// TIA Portal V15.1 export
// export: Created 2024-05-17T05:38:21.4668831Z, ExportSetting WithDefaults, DisplayName Totally Integrated Automation Portal, DisplayVersion V15.1 Update 5, DisplayName TIA Portal Openness, DisplayVersion V15.1 Update 5, DisplayName SINAMICS Startdrive Advanced, DisplayVersion V15.1, DisplayName G130, G150, S120, S150, SINAMICS MV, S210, DisplayVersion V15.1, DisplayName G110M, G120, G120C, G120D, G120P, DisplayVersion V15.1, DisplayName STEP 7 Professional, DisplayVersion V15.1 Update 5, DisplayName STEP 7 Safety, DisplayVersion V15.1, DisplayName WinCC Professional, DisplayVersion V15.1 Update 5, DisplayName SIMATIC Visualization Architect, DisplayVersion V15.1
DATA_BLOCK "_209220CS22"   // DB1845
{ S7_Optimized_Access := 'TRUE' }
VERSION : 0.1
// stored: AutoNumber false, DBAccessibleFromOPCUA true, InstanceOfName LGBLineConvBrake-MDXPN-DFS22B, InstanceOfType FB
"LGBLineConvBrake-MDXPN-DFS22B"
   // VAR_INPUT
   //    I_DetArrived { ExternalAccessible := 'False'; ExternalVisible := 'False'; ExternalWritable := 'False'} : Bool;
   //    I_DetSaturation { ExternalAccessible := 'False'; ExternalVisible := 'False'; ExternalWritable := 'False'} : Bool;
   //    I_DetMinGapLeft { ExternalAccessible := 'False'; ExternalVisible := 'False'; ExternalWritable := 'False'} : Bool;
   //    I_DetMinGapRight { ExternalAccessible := 'False'; ExternalVisible := 'False'; ExternalWritable := 'False'} : Bool;
   //    I_DetBeltTension { ExternalAccessible := 'False'; ExternalVisible := 'False'; ExternalWritable := 'False'} : Bool;
   //    I_TrfInSetBegin { ExternalAccessible := 'False'; ExternalVisible := 'False'; ExternalWritable := 'False'} : Bool;
   //    I_TrfInSetIntlkOk { ExternalAccessible := 'False'; ExternalVisible := 'False'; ExternalWritable := 'False'} : Bool;
   //    I_TrfInSetRdyDlv { ExternalAccessible := 'False'; ExternalVisible := 'False'; ExternalWritable := 'False'} : Bool;
   //    I_TrfInSetTM { ExternalAccessible := 'False'; ExternalVisible := 'False'; ExternalWritable := 'False'} : Bool;
   //    I_TrfOutSetBegin { ExternalAccessible := 'False'; ExternalVisible := 'False'; ExternalWritable := 'False'} : Bool;
   //    I_TrfOutSetIntlkOk { ExternalAccessible := 'False'; ExternalVisible := 'False'; ExternalWritable := 'False'} : Bool;
   //    I_TrfOutSetRdyRcv { ExternalAccessible := 'False'; ExternalVisible := 'False'; ExternalWritable := 'False'} : Bool;
   //    I_TrfOutSetArrived { ExternalAccessible := 'False'; ExternalVisible := 'False'; ExternalWritable := 'False'} : Bool;
   //    I_StopProduction { ExternalAccessible := 'False'; ExternalVisible := 'False'; ExternalWritable := 'False'} : Bool;
   //    I_ExtStopCondition { ExternalAccessible := 'False'; ExternalVisible := 'False'; ExternalWritable := 'False'} : Bool;
   //    I_InfeedBegin { ExternalAccessible := 'False'; ExternalVisible := 'False'; ExternalWritable := 'False'} : Bool;
   //    I_ManInfeedAllowed { ExternalAccessible := 'False'; ExternalVisible := 'False'; ExternalWritable := 'False'} : Bool;
   //    I_EnabledriveCon { ExternalAccessible := 'False'; ExternalVisible := 'False'; ExternalWritable := 'False'} : Bool;
   //    I_FreeRunningBrakeDriveCon { ExternalAccessible := 'False'; ExternalVisible := 'False'; ExternalWritable := 'False'} : Bool;
   //    I_MotorProtection { ExternalAccessible := 'False'; ExternalVisible := 'False'; ExternalWritable := 'False'} : Bool;
   //    I_BrakeProtection { ExternalAccessible := 'False'; ExternalVisible := 'False'; ExternalWritable := 'False'} : Bool;
   //    I_SafetySwitchMotPower { ExternalAccessible := 'False'; ExternalVisible := 'False'; ExternalWritable := 'False'} : Bool;
   //    I_SafetySwitchMotBrake { ExternalAccessible := 'False'; ExternalVisible := 'False'; ExternalWritable := 'False'} : Bool;
   //    I_ReverseKeySwitch1 { ExternalAccessible := 'False'; ExternalVisible := 'False'; ExternalWritable := 'False'} : Bool;
   //    I_ReverseKeySwitch2 { ExternalAccessible := 'False'; ExternalVisible := 'False'; ExternalWritable := 'False'} : Bool;
   //    I_LocalPBSet { ExternalAccessible := 'False'; ExternalVisible := 'False'; ExternalWritable := 'False'} : Bool;
   //    I_LocalPBRes { ExternalAccessible := 'False'; ExternalVisible := 'False'; ExternalWritable := 'False'} : Bool;
   //    I_LocalPBSetMotPower { ExternalAccessible := 'False'; ExternalVisible := 'False'; ExternalWritable := 'False'} : Bool;
   //    I_LocalPBResMotPower { ExternalAccessible := 'False'; ExternalVisible := 'False'; ExternalWritable := 'False'} : Bool;
   //    I_LocalPBSetMotBrake { ExternalAccessible := 'False'; ExternalVisible := 'False'; ExternalWritable := 'False'} : Bool;
   //    I_LocalPBResMotBrake { ExternalAccessible := 'False'; ExternalVisible := 'False'; ExternalWritable := 'False'} : Bool;
   //    I_SafetyOk { ExternalAccessible := 'False'; ExternalVisible := 'False'; ExternalWritable := 'False'} : Bool;
   //    I_MotionStopOk { ExternalAccessible := 'False'; ExternalVisible := 'False'; ExternalWritable := 'False'} : Bool;
   //    I_Torque { ExternalAccessible := 'False'; ExternalVisible := 'False'; ExternalWritable := 'False'} : Int;
   //    I_Speed { ExternalAccessible := 'False'; ExternalVisible := 'False'; ExternalWritable := 'False'} : Int;
   //    I_SpeedHandHeld { ExternalAccessible := 'False'; ExternalVisible := 'False'; ExternalWritable := 'False'} : Int;
   //    I_HandHeldSelected { ExternalAccessible := 'False'; ExternalVisible := 'False'; ExternalWritable := 'False'} : Bool;
   //    I_SafetyStatusWordMotPower1 { ExternalAccessible := 'False'; ExternalVisible := 'False'; ExternalWritable := 'False'} : Word;
   //    I_SafetyStatusWordMotPower2 { ExternalAccessible := 'False'; ExternalVisible := 'False'; ExternalWritable := 'False'} : Word;
   //    I_SafetyStatusWordMotPower3 { ExternalAccessible := 'False'; ExternalVisible := 'False'; ExternalWritable := 'False'} : Word;
   //    I_SafetyControlWordMotPower1 { ExternalAccessible := 'False'; ExternalVisible := 'False'; ExternalWritable := 'False'} : Word;
   //    I_SafetyControlWordMotPower2 { ExternalAccessible := 'False'; ExternalVisible := 'False'; ExternalWritable := 'False'} : Word;
   //    I_SafetyControlWordMotPower3 { ExternalAccessible := 'False'; ExternalVisible := 'False'; ExternalWritable := 'False'} : Word;
   //    I_SafetyStatusWordBrakeMotor { ExternalAccessible := 'False'; ExternalVisible := 'False'; ExternalWritable := 'False'} : Word;
   //    I_SafetyControlWordBrakeMotor { ExternalAccessible := 'False'; ExternalVisible := 'False'; ExternalWritable := 'False'} : Word;
   // END_VAR
   // VAR_OUTPUT
   //    O_Active { ExternalAccessible := 'False'; ExternalVisible := 'False'; ExternalWritable := 'False'} : Bool;
   //    O_ActiveMotPower { ExternalAccessible := 'False'; ExternalVisible := 'False'; ExternalWritable := 'False'} : Bool;
   //    O_ActiveMotBrake { ExternalAccessible := 'False'; ExternalVisible := 'False'; ExternalWritable := 'False'} : Bool;
   //    O_ReadyForOperation { ExternalAccessible := 'False'; ExternalVisible := 'False'; ExternalWritable := 'False'} : Bool;
   //    O_TrfInSetRdyRcv { ExternalAccessible := 'False'; ExternalVisible := 'False'; ExternalWritable := 'False'} : Bool;
   //    O_TrfInSetArrived { ExternalAccessible := 'False'; ExternalVisible := 'False'; ExternalWritable := 'False'} : Bool;
   //    O_TrfInSetActive { ExternalAccessible := 'False'; ExternalVisible := 'False'; ExternalWritable := 'False'} : Bool;
   //    O_TrfInSetFinished { ExternalAccessible := 'False'; ExternalVisible := 'False'; ExternalWritable := 'False'} : Bool;
   //    O_TrfOutSetRdyDlv { ExternalAccessible := 'False'; ExternalVisible := 'False'; ExternalWritable := 'False'} : Bool;
   //    O_TrfOutSetTM { ExternalAccessible := 'False'; ExternalVisible := 'False'; ExternalWritable := 'False'} : Bool;
   //    O_TrfOutSetActive { ExternalAccessible := 'False'; ExternalVisible := 'False'; ExternalWritable := 'False'} : Bool;
   //    O_TrfOutSetFinished { ExternalAccessible := 'False'; ExternalVisible := 'False'; ExternalWritable := 'False'} : Bool;
   //    O_Saturation { ExternalAccessible := 'False'; ExternalVisible := 'False'; ExternalWritable := 'False'} : Bool;
   //    O_EcoMode { ExternalAccessible := 'False'; ExternalVisible := 'False'; ExternalWritable := 'False'} : Bool;
   //    O_LedRoller { ExternalAccessible := 'False'; ExternalVisible := 'False'; ExternalWritable := 'False'} : Bool;
   //    O_EnableDriveMotPower { ExternalAccessible := 'False'; ExternalVisible := 'False'; ExternalWritable := 'False'} : Bool;
   //    O_EnableDriveMotBrake { ExternalAccessible := 'False'; ExternalVisible := 'False'; ExternalWritable := 'False'} : Bool;
   //    O_ResetBrakeDrive { ExternalAccessible := 'False'; ExternalVisible := 'False'; ExternalWritable := 'False'} : Bool;
   //    O_FreeRunningBrakeDrive { ExternalAccessible := 'False'; ExternalVisible := 'False'; ExternalWritable := 'False'} : Bool;
   //    O_AlarmABCondition { ExternalAccessible := 'False'; ExternalVisible := 'False'; ExternalWritable := 'False'} : Bool;
   //    O_AlarmA { ExternalAccessible := 'False'; ExternalVisible := 'False'; ExternalWritable := 'False'} : Bool;
   //    O_AlarmB { ExternalAccessible := 'False'; ExternalVisible := 'False'; ExternalWritable := 'False'} : Bool;
   //    O_AlarmC { ExternalAccessible := 'False'; ExternalVisible := 'False'; ExternalWritable := 'False'} : Bool;
   //    O_AlarmD { ExternalAccessible := 'False'; ExternalVisible := 'False'; ExternalWritable := 'False'} : Bool;
   //    H_AlarmWord { ExternalAccessible := 'False'; ExternalVisible := 'False'; ExternalWritable := 'False'} : DWord;
   // END_VAR
   // VAR_IN_OUT
   //    IO_Modes : "Modes";
   //    H_HMI : "H_HMI";
   //    "H_GBLineConvBrake-MDXPN-DFS22B" : "H_GBLineConvBrake-MDXPN-DFS22B";
   //    C_Config : "LineConvBrake-MDXPNConfig";
   // END_VAR
   // VAR
   //    AA_MotorProtection { ExternalAccessible := 'False'; ExternalVisible := 'False'; ExternalWritable := 'False'} : Bool;
   //    AA_BrakeProtection { ExternalAccessible := 'False'; ExternalVisible := 'False'; ExternalWritable := 'False'} : Bool;
   //    AA_SafetySwitchMotPower { ExternalAccessible := 'False'; ExternalVisible := 'False'; ExternalWritable := 'False'} : Bool;
   //    AA_SafetySwitchMotBrake { ExternalAccessible := 'False'; ExternalVisible := 'False'; ExternalWritable := 'False'} : Bool;
   //    AB_AlarmMotPower { ExternalAccessible := 'False'; ExternalVisible := 'False'; ExternalWritable := 'False'} : Bool;
   //    AB_MinGapLeft { ExternalAccessible := 'False'; ExternalVisible := 'False'; ExternalWritable := 'False'} : Bool;
   //    AB_MinGapRight { ExternalAccessible := 'False'; ExternalVisible := 'False'; ExternalWritable := 'False'} : Bool;
   //    AB_TrfOutSetOverTime { ExternalAccessible := 'False'; ExternalVisible := 'False'; ExternalWritable := 'False'} : Bool;
   //    AC_TrfInStopped { ExternalAccessible := 'False'; ExternalVisible := 'False'; ExternalWritable := 'False'} : Bool;
   //    AC_MinGapLeft { ExternalAccessible := 'False'; ExternalVisible := 'False'; ExternalWritable := 'False'} : Bool;
   //    AC_MinGapRight { ExternalAccessible := 'False'; ExternalVisible := 'False'; ExternalWritable := 'False'} : Bool;
   //    AC_BeltTension { ExternalAccessible := 'False'; ExternalVisible := 'False'; ExternalWritable := 'False'} : Bool;
   //    AD_WarningMotPower { ExternalAccessible := 'False'; ExternalVisible := 'False'; ExternalWritable := 'False'} : Bool;
   //    AD_WarningMotBrake { ExternalAccessible := 'False'; ExternalVisible := 'False'; ExternalWritable := 'False'} : Bool;
   //    AD_TrfOutSetInterlock { ExternalAccessible := 'False'; ExternalVisible := 'False'; ExternalWritable := 'False'} : Bool;
   //    AD_TrfInSetInterlock { ExternalAccessible := 'False'; ExternalVisible := 'False'; ExternalWritable := 'False'} : Bool;
   //    AD_SaturationState { ExternalAccessible := 'False'; ExternalVisible := 'False'; ExternalWritable := 'False'} : Bool;
   //    AD_MotionStop { ExternalAccessible := 'False'; ExternalVisible := 'False'; ExternalWritable := 'False'} : Bool;
   //    AC_ConfigCalibrationAlm { ExternalAccessible := 'False'; ExternalVisible := 'False'; ExternalWritable := 'False'} : Bool;
   //    AD_CalibrationSetWarn { ExternalAccessible := 'False'; ExternalVisible := 'False'; ExternalWritable := 'False'} : Bool;
   //    AC_ConfigRampAlmMotPower { ExternalAccessible := 'False'; ExternalVisible := 'False'; ExternalWritable := 'False'} : Bool;
   //    AC_ConfigRampCalcAlmMotPower { ExternalAccessible := 'False'; ExternalVisible := 'False'; ExternalWritable := 'False'} : Bool;
   //    AC_ConfigRampAlmMotBrake { ExternalAccessible := 'False'; ExternalVisible := 'False'; ExternalWritable := 'False'} : Bool;
   //    AC_ConfigRampCalcAlmMotBrake { ExternalAccessible := 'False'; ExternalVisible := 'False'; ExternalWritable := 'False'} : Bool;
   //    AA_NoBusControlMotBrake { ExternalAccessible := 'False'; ExternalVisible := 'False'; ExternalWritable := 'False'} : Bool;
   //    PODataNotEnabled { ExternalAccessible := 'False'; ExternalVisible := 'False'; ExternalWritable := 'False'} : Bool;
   //    SafetyOk { ExternalAccessible := 'False'; ExternalVisible := 'False'; ExternalWritable := 'False'} : Bool;
   //    TrfInfeedHoldSet { ExternalAccessible := 'False'; ExternalVisible := 'False'; ExternalWritable := 'False'} : Bool;
   //    TrfOutSetCmd { ExternalAccessible := 'False'; ExternalVisible := 'False'; ExternalWritable := 'False'} : Bool;
   //    TrfOutfeedHoldSet { ExternalAccessible := 'False'; ExternalVisible := 'False'; ExternalWritable := 'False'} : Bool;
   //    TrfInSetCmd { ExternalAccessible := 'False'; ExternalVisible := 'False'; ExternalWritable := 'False'} : Bool;
   //    TrfInSetActive { ExternalAccessible := 'False'; ExternalVisible := 'False'; ExternalWritable := 'False'} : Bool;
   //    TrfOutSetActive { ExternalAccessible := 'False'; ExternalVisible := 'False'; ExternalWritable := 'False'} : Bool;
   //    TrfOutSetFinished { ExternalAccessible := 'False'; ExternalVisible := 'False'; ExternalWritable := 'False'} : Bool;
   //    TrfOutSetRdyDlv { ExternalAccessible := 'False'; ExternalVisible := 'False'; ExternalWritable := 'False'} : Bool;
   //    TrfOutSetTM { ExternalAccessible := 'False'; ExternalVisible := 'False'; ExternalWritable := 'False'} : Bool;
   //    TrfInSetRdyRcv { ExternalAccessible := 'False'; ExternalVisible := 'False'; ExternalWritable := 'False'} : Bool;
   //    TrfInSetArrived { ExternalAccessible := 'False'; ExternalVisible := 'False'; ExternalWritable := 'False'} : Bool;
   //    TrfInSetFinished { ExternalAccessible := 'False'; ExternalVisible := 'False'; ExternalWritable := 'False'} : Bool;
   //    TrfOutSetAlmCond { ExternalAccessible := 'False'; ExternalVisible := 'False'; ExternalWritable := 'False'} : Bool;
   //    TrfInSetTrfOutSetTM { ExternalAccessible := 'False'; ExternalVisible := 'False'; ExternalWritable := 'False'} : Bool;
   //    MotorcmdHspdSetMotPower { ExternalAccessible := 'False'; ExternalVisible := 'False'; ExternalWritable := 'False'} : Bool;
   //    MotorcmdHspdResMotPower { ExternalAccessible := 'False'; ExternalVisible := 'False'; ExternalWritable := 'False'} : Bool;
   //    MotorcmdHspdSetMotBrake { ExternalAccessible := 'False'; ExternalVisible := 'False'; ExternalWritable := 'False'} : Bool;
   //    MotorcmdHspdResMotBrake { ExternalAccessible := 'False'; ExternalVisible := 'False'; ExternalWritable := 'False'} : Bool;
   //    MotCmdAutoCond { ExternalAccessible := 'False'; ExternalVisible := 'False'; ExternalWritable := 'False'} : Bool;
   //    StationOnly { ExternalAccessible := 'False'; ExternalVisible := 'False'; ExternalWritable := 'False'} : Bool;
   //    AlarmA { ExternalAccessible := 'False'; ExternalVisible := 'False'; ExternalWritable := 'False'} : Bool;
   //    AlarmB { ExternalAccessible := 'False'; ExternalVisible := 'False'; ExternalWritable := 'False'} : Bool;
   //    AlarmC { ExternalAccessible := 'False'; ExternalVisible := 'False'; ExternalWritable := 'False'} : Bool;
   //    AlarmD { ExternalAccessible := 'False'; ExternalVisible := 'False'; ExternalWritable := 'False'} : Bool;
   //    AlarmABCondition { ExternalAccessible := 'False'; ExternalVisible := 'False'; ExternalWritable := 'False'} : Bool;
   //    MinGapLeftAlmCond { ExternalAccessible := 'False'; ExternalVisible := 'False'; ExternalWritable := 'False'} : Bool;
   //    MinGapRightAlmCond { ExternalAccessible := 'False'; ExternalVisible := 'False'; ExternalWritable := 'False'} : Bool;
   //    ReadyForOperationMotPower { ExternalAccessible := 'False'; ExternalVisible := 'False'; ExternalWritable := 'False'} : Bool;
   //    ReadyForOperationMotBrake { ExternalAccessible := 'False'; ExternalVisible := 'False'; ExternalWritable := 'False'} : Bool;
   //    MotorLoopActiveMotPower { ExternalAccessible := 'False'; ExternalVisible := 'False'; ExternalWritable := 'False'} : Bool;
   //    MotorLoopActiveMotBrake { ExternalAccessible := 'False'; ExternalVisible := 'False'; ExternalWritable := 'False'} : Bool;
   //    MotorLoopAlarmCondMotPower { ExternalAccessible := 'False'; ExternalVisible := 'False'; ExternalWritable := 'False'} : Bool;
   //    MotorLoopAlarmCondMotBrake { ExternalAccessible := 'False'; ExternalVisible := 'False'; ExternalWritable := 'False'} : Bool;
   //    PulsInfeedBegin { ExternalAccessible := 'False'; ExternalVisible := 'False'; ExternalWritable := 'False'} : Bool;
   //    MaxTimeResetDirection { ExternalAccessible := 'False'; ExternalVisible := 'False'; ExternalWritable := 'False'} : Bool;
   //    LineConveyorEmpty { ExternalAccessible := 'False'; ExternalVisible := 'False'; ExternalWritable := 'False'} : Bool;
   //    LineConveyorEmptyTime { ExternalAccessible := 'False'; ExternalVisible := 'False'; ExternalWritable := 'False'} : DInt;
   //    ResetDirectionTime { ExternalAccessible := 'False'; ExternalVisible := 'False'; ExternalWritable := 'False'} : DInt;
   //    Speed { ExternalAccessible := 'False'; ExternalVisible := 'False'; ExternalWritable := 'False'} : Int;
   //    DummyReal { ExternalAccessible := 'False'; ExternalVisible := 'False'; ExternalWritable := 'False'} : Real;
   //    Edge { ExternalAccessible := 'False'; ExternalVisible := 'False'; ExternalWritable := 'False'} : Array[1..10] of Bool;
   //    _LTrfInSet { ExternalAccessible := 'False'; ExternalVisible := 'False'; ExternalWritable := 'False'} : "LGBChainTrfIn";
   //    _LTrfOutSet { ExternalAccessible := 'False'; ExternalVisible := 'False'; ExternalWritable := 'False'} : "LGBTrfOut";
   //    _LineConvMotPower { ExternalAccessible := 'False'; ExternalVisible := 'False'; ExternalWritable := 'False'} : "LGBMotor2W2S-MDXPN-6PD-DFS22B";
   //    _LineConvMotBrake { ExternalAccessible := 'False'; ExternalVisible := 'False'; ExternalWritable := 'False'} : "LGBMotorTorque-MDXPN-3PD";
   //    _CheckMinGapLeft { ExternalAccessible := 'False'; ExternalVisible := 'False'; ExternalWritable := 'False'} : "L1AlarmMultiIn";
   //    _CheckMinGapRight { ExternalAccessible := 'False'; ExternalVisible := 'False'; ExternalWritable := 'False'} : "L1AlarmMultiIn";
   //    _Check2MinGapLeft { ExternalAccessible := 'False'; ExternalVisible := 'False'; ExternalWritable := 'False'} : "L1AlarmMultiIn";
   //    _Check2MinGapRight { ExternalAccessible := 'False'; ExternalVisible := 'False'; ExternalWritable := 'False'} : "L1AlarmMultiIn";
   //    _CheckBeltTension { ExternalAccessible := 'False'; ExternalVisible := 'False'; ExternalWritable := 'False'} : "L1AlarmMultiIn";
   //    _StationOnly { ExternalAccessible := 'False'; ExternalVisible := 'False'; ExternalWritable := 'False'} : "LToggle";
   //    _NoTrfIn { ExternalAccessible := 'False'; ExternalVisible := 'False'; ExternalWritable := 'False'} : "LToggle";
   //    _Saturation { ExternalAccessible := 'False'; ExternalVisible := 'False'; ExternalWritable := 'False'} : IEC_TIMER;
   //    _MaxTimeResetDirection { ExternalAccessible := 'False'; ExternalVisible := 'False'; ExternalWritable := 'False'} : IEC_TIMER;
   //    _EcoMode { ExternalAccessible := 'False'; ExternalVisible := 'False'; ExternalWritable := 'False'} : IEC_TIMER;
   // END_VAR
BEGIN
END_DATA_BLOCK
